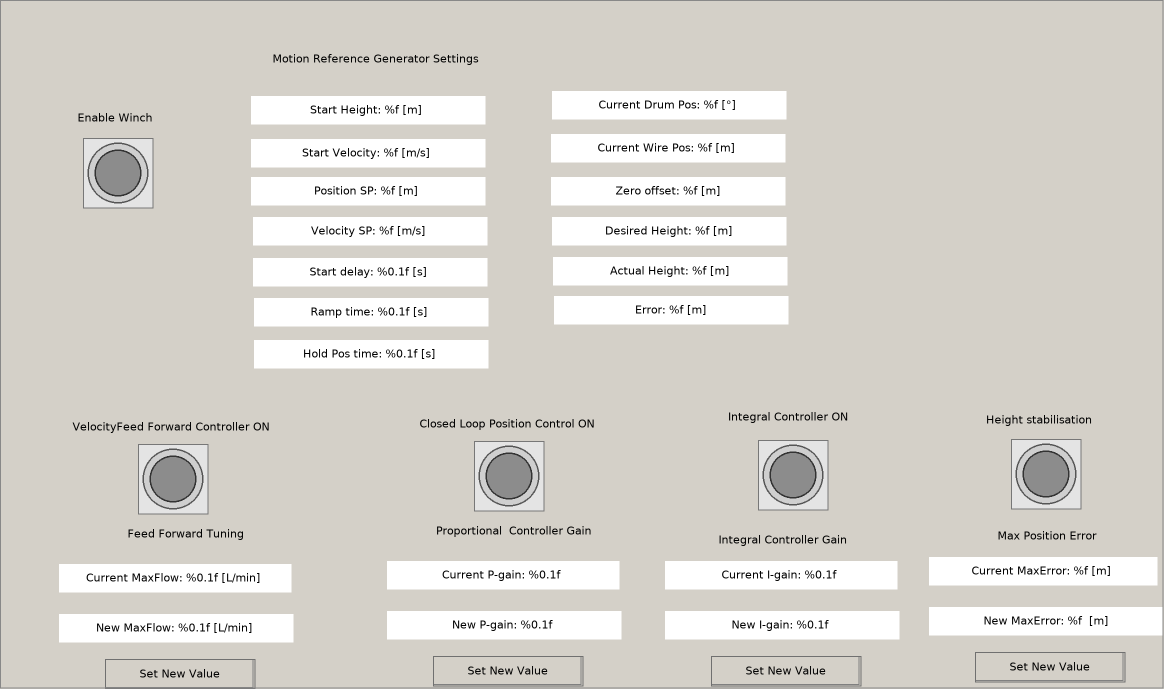
VISUALIZATION Winch  // 1164x689
    Label (40,103 150x30), "Enable Winch"
    PushSwitch (83,138 70x70), variable: G_Hmi.bWinchEnable, behaviour: TOGGLE, style: Switch-PushSwitch-Gray
    Label (230,44 291x30), "Motion Reference Generator Settings"
    Textfield (250,95 236x30), "Start Height: %f [m]", text variable: G_Hmi.stMotionReferenceGeneratorSettingsWinch.fStartPosition_m
        OnMouseDown: write the text variable via Default, min 0, max 1.0
    Textfield (250,138 236x30), "Start Velocity: %f [m/s]", text variable: G_Hmi.stMotionReferenceGeneratorSettingsWinch.fStartVelocity_m
        OnMouseDown: write the text variable via Default, min 0, max 0.05
    Textfield (250,176 236x30), "Position SP: %f [m]", text variable: G_Hmi.stMotionReferenceGeneratorSettingsWinch.fPositionSetpoint_ms
        OnMouseDown: write the text variable via Default, min 0, max 1.0
    Textfield (252,216 236x30), "Velocity SP: %f [m/s]", text variable: G_Hmi.stMotionReferenceGeneratorSettingsWinch.fVelocitySetpoint_m
        OnMouseDown: write the text variable via Default, min 0, max 0.05
    Textfield (252,257 236x30), "Start delay: %0.1f [s]", text variable: G_Hmi.stMotionReferenceGeneratorSettingsWinch.fTimeBeforeStarting_s
        OnMouseDown: write the text variable via Default, min 0, max 10
    Textfield (253,297 236x30), "Ramp time: %0.1f [s]", text variable: G_Hmi.stMotionReferenceGeneratorSettingsWinch.fRampTime_s
        OnMouseDown: write the text variable via Default, min 0, max 10
    Textfield (253,339 236x30), "Hold Pos time: %0.1f [s]", text variable: G_Hmi.stMotionReferenceGeneratorSettingsWinch.fHoldPositionTime_s
        OnMouseDown: write the text variable via Default, min 0, max 10
    Textfield (551,90 236x30), "Current Drum Pos: %f [°]", text variable: G_Sensors.fWinchEncoderPosition
        OnMouseDown: write the text variable via Default, min 0, max 0.5
    Button (433,656 150x30), "Set New Value"
        tap G_Hmi.stModifyAutomaticControlSettingsWinch.bSetNewProportionalGain
    Textfield (386,560 234x30), "Current P-gain: %0.1f", text variable: G_Parameters.stParam.stClosedLoopControlSettingsWinch.fProportionalGain
    Textfield (386,610 236x30), "New P-gain: %0.1f", text variable: G_Hmi.stModifyAutomaticControlSettingsWinch.fNewProportionalGain
        OnMouseDown: write the text variable via Default
    Label (431,516 166x30), "Proportional Controller Gain"
    Button (711,656 150x30), "Set New Value"
        tap G_Hmi.stModifyAutomaticControlSettingsWinch.bSetNewIntegralGain
    Textfield (664,560 234x30), "Current I-gain: %0.1f", text variable: G_Parameters.stParam.stClosedLoopControlSettingsWinch.fIntegralGain
    Textfield (664,610 236x30), "New I-gain: %0.1f", text variable: G_Hmi.stModifyAutomaticControlSettingsWinch.fNewIntegralGain
        OnMouseDown: write the text variable via Default
    Label (708,525 150x30), "Integral Controller Gain"
    PushSwitch (758,440 70x70), variable: G_Hmi.stAutomaticControlSettingsWinch.bEnableIntegralController, behaviour: TOGGLE, style: Switch-PushSwitch-Gray
    Label (705,402 166x30), "Integral Controller ON"
    Label (381,409 252x30), "Closed Loop Position Control ON"
    PushSwitch (474,441 70x70), variable: G_Hmi.stAutomaticControlSettingsWinch.bEnableClosedLoopPositionControl, behaviour: TOGGLE, style: Switch-PushSwitch-Gray
    Label (45,412 252x30), "VelocityFeed Forward Controller ON"
    PushSwitch (138,444 70x70), variable: G_Hmi.stAutomaticControlSettingsWinch.bEnableVelocityFeedForwardControl, behaviour: TOGGLE, style: Switch-PushSwitch-Gray
    Button (105,659 150x30), "Set New Value"
        tap G_Hmi.stModifyAutomaticControlSettingsWinch.bSetNewMaxFlowCapacity p1329445385=TRUE
    Textfield (58,563 234x30), "Current MaxFlow: %0.1f [L/min]", text variable: G_Parameters.stParam.stOpenLoopControlSettingsWinch.fMaxFlowCapacity
    Textfield (58,613 236x30), "New MaxFlow: %0.1f [L/min]", text variable: G_Hmi.stModifyAutomaticControlSettingsWinch.fNewMaxFlowCapacity
        OnMouseDown: write the text variable via Default, min 0.0001, max 100
    Label (103,519 166x30), "Feed Forward Tuning"
    Button (975,652 150x30), "Set New Value"
        tap G_Hmi.stModifyAutomaticControlSettingsWinch.bSetNewMaxPositionError
    Textfield (928,556 230x30), "Current MaxError: %f [m]", text variable: G_Parameters.stParam.stClosedLoopControlSettingsWinch.fMaxPositionError
    Textfield (928,606 236x30), "New MaxError: %f [m]", text variable: G_Hmi.stModifyAutomaticControlSettingsWinch.fNewMaxPositionError
        OnMouseDown: write the text variable via Default
    Label (972,521 150x30), "Max Position Error"
    Textfield (550,133 236x30), "Current Wire Pos: %f [m]", text variable: G_Sensors.fWinchWirePosition
        OnMouseDown: write the text variable via Default, min 0, max 0.5
    PushSwitch (1011,439 70x70), variable: G_HeightCorrection.xCorrectHeight, behaviour: TOGGLE, style: Switch-PushSwitch-Gray
    Label (956,405 166x30), "Height stabilisation"
    Textfield (550,176 236x30), "Zero offset: %f [m]", text variable: G_HeightCorrection.rZeroOffset
        OnMouseDown: write the text variable via Default, min -100.0, max 100.0
    Textfield (551,216 236x30), "Desired Height: %f [m]", text variable: G_HeightCorrection.rDesiredHeight
        OnMouseDown: write the text variable via Default, min 0, max 0.5
    Textfield (552,256 236x30), "Actual Height: %f [m]", text variable: G_HeightCorrection.rActual
        OnMouseDown: write the text variable via Default, min 0, max 0.5
    Textfield (553,295 236x30), "Error: %f [m]", text variable: G_Sensors.fWinchWirePosition
        OnMouseDown: write the text variable via Default, min 0, max 0.5
END_VISUALIZATION

(* stored: Version 1.1.0.1, ProductVersion 3.1.4024.11
   Visu Winch: Id {d4968b97-4ba6-4a28-b2f2-fd4f65046f3b} *)
